Staubli VAL3: isInSafetyArea.pgx

program isInSafetyArea()
  local jointRs l_jHere
  local num l_ns
  local pointRs l_pCurrent
begin
  bIsConnectPC=false
  do
    l_pCurrent=here(flange,world)
    //**************************************************//
    //******** 用来判断机器人是否在安全工作空间 ********//
    //**************************************************//
    if (l_pCurrent.trsf.y>=nSafeMaxY or l_pCurrent.trsf.y<=nSafeMinY or l_pCurrent.trsf.x>=nSafeMaxX or l_pCurrent.trsf.x<=nSafeMinX) and _nOmacStat==3
      aioSet(aRbAlarm,10)
      call setAlarm(7)
      popUpMsg("机器人超出安全工作空间！")
      logMsg("机器人超出安全工作空间！")
      call OMAC_Abort()
    endIf

    if (dConvControl[0]==true)
      dConvControl[1]=true
    else
      dConvControl[1]=false
    endIf

    if (bIsConnectPC==true)
      if (sDataPC=="stop")
        l_ns=clock()
        do
          call setAlarm(0)
        until (clock()-l_ns>0.5)
        call setAlarm(10)
        sDataPC="alarm0"
        bIsConnectPC=false
      endIf
    endIf
    delay(0)
  until false
end
